// TIA Portal V19 export
FUNCTION "AutoAndResetTank" : Void   // FC56, STL
TITLE = Reset UHT
{ S7_Optimized_Access := 'TRUE' }
AUTHOR : OPA_8160
NAME : RESET
VERSION : 0.2
// ****** REVISION HISTORY :
// 
// VERSION DATE       BY  DESCRIPTION
// --------------------------------------------------------------------------
// 00.00               ORIGINAL FUNCTION BLOCK
// 
// 00.01 10/12 1997   OPA
//       FOLLOWING INSTRUCTIONS HAVE BEEN ADDED IN NETWORK 6
//       R     "S.T.01.REQUEST LYE"   "M242.0"     // STOP REQUESTING DETERGENT
//       R     "S.T.01.REQUEST ACID"  "M242.1"     // STOP REQUESTING DETERGENT
//       WITHOUT THESE TWO INSTRUCTIONS, DETERGENT PUMPS (LYE/ACID) COULD
//       CONTINUE DOSING AFTER STOP. 
// 00.02 11/2 1998    OPA   "S0 STOP CIP TANK" ADDED FOR "TANK AUTO"
// stored: AutoNumber false
BEGIN

NETWORK
TITLE = SET AUTO FLAG TANK
      O     "S0 PRESTERILIZING";
      O     "S0 STOP PRESTE. TANK";
      O     "S0 PRODUCTION TANK";
      O     "S0 STOP PRODUCTION TANK";
      O     "S0 CIP TANK";
      O     "S0 STOP CIP TANK";
      O     "S0 TOTAL STOP TANK";
      O     "LEDAssignment".SPARE_BUTTON1;

      =     "TANK AUTO";
      A     "LEDAssignment".SPARE_BUTTON1;

      R     "LEDAssignment".SPARE_BUTTON1;
      AN    "TANK AUTO";
      =     "M_AHV_SHUT_DOWN";
      AN    "S0 CIP TANK";
      JC    M001;
      A     "LowCIPPressure";
      JC    M003;  //"DB SETPOINTS".PT0167SpCIP
      A     "AcidCipPressure";
      JC    M004;
      L     "Setpoints".PT0167SpCIP;  // "DB SETPOINTS".PT0167SpCIPLow
      T     "STP_PT0167/IP0149_50".PT0167SpSTP;
      JU    M001;
M003: L     "Setpoints".PT0167SpCIPLow;
      T     "STP_PT0167/IP0149_50".PT0167SpSTP;
      JU    M001;
M004: L     "Setpoints".PT0167AcidPressure;
      T     "STP_PT0167/IP0149_50".PT0167SpSTP;

NETWORK
TITLE = FORCE VALVES TO AUTO
// THIS FORCE FUNCTION SETS ALL OUTPUTS IN AUTO MODE. I.E. VALVES, MOTORS, PUMPS 
// ETC.
M001: A     "TANK AUTO";
      FP    "ForceValves";
      JNB   M002;
      CALL  "Output Force to auto";
M002: NOP   0;

NETWORK
TITLE = RESET MANUAL MODE ON REGULATORS
// MAKE SURE THAT ALL RESET FROM AUTO, MANUAL, CASCADE OR FIXED MODE WHEN THE 
// PLANT 
// ENTER AUTO MODE
      AN    "TANK AUTO";
      FP    "UnforceValves";
      R     "AutoTT0172/IP0157";
      R     "ManTT0172/IP0157";
      R     "AutoPT0167/IP0149";
      R     "ManPT0167/IP0149";

NETWORK
TITLE = SET DUMMY RESET TANK
// THE FOLLOWING NETWORKS WILL RESET THE UHT-PLANT IF THE "UHT AUTO" FLAG 
// DISAPPEARS!
// I.E. PREPARE TOTAL STOP
      A     "TANK AUTO";
      S     "DUMMY RESET TANK";
      BEC;
      AN    "DUMMY RESET TANK";
      BEC;
      R     "DUMMY RESET TANK";

NETWORK
TITLE = RESET MAIN FLAGS FOR ALL DIFFERENT TANK-PROGRAM STEPS
      SET;
      R     "S0 STOP PRESTE. TANK";
      R     "S0 PRESTERILIZING";
      R     "S0 PRODUCTION TANK";
      R     "S0 STOP PRODUCTION TANK";
      R     "S0 TOTAL STOP TANK";
      R     "S0 CIP TANK";
      R     "S16 CIP TANK";

NETWORK
TITLE = RESET LED'S ON OPERATORPANEL
      R     "TANK STERILE";
      R     "TANK INITIALIZED";
      R     "LEDAssignment".K1_FLASH;  //"FLASH_K1_SPARE"
      R     "LEDAssignment".K1_LIGHT;  //"LIGHT_K1_SPARE"
      R     "LEDAssignment".K2_FLASH;  //"FLASH_K2_SPARE"
      R     "LEDAssignment".K2_LIGHT;  //"LIGHT_K2_SPARE"
      R     "LEDAssignment".K3_FLASH;  //"FLASH_K3_PRESTE."
      R     "LEDAssignment".K3_LIGHT;  //"LIGHT_K3_PRESTE."
      R     "LEDAssignment".K4_FLASH;  //"FLASH_K4_CIP_LYE"
      R     "LEDAssignment".K4_LIGHT;  //"LIGHT_K4_CIP_LYE"
      R     "LEDAssignment".K5_FLASH;  //"FLASH_K5_CIP_LYE_ACID"
      R     "LEDAssignment".K5_LIGHT;  //"LIGHT_K5_CIP_LYE_ACID"
      R     "LEDAssignment".K6_FLASH;  //"FLASH_K6_DRAIN_TANK"
      R     "LEDAssignment".K6_LIGHT;  //"LIGHT_K6_DRAIN_TANK"
      R     "LEDAssignment".K7_FLASH;  //"FLASH_K7_STOP"
      R     "LEDAssignment".K7_LIGHT;  //"LIGHT_K7_STOP"
//      R     M     57.6
//      R     M     57.7
      L     2#0000_0000_0000_0000;
//      T     MW    48                    // F-PUSHBUTTONS
//      T     MW    50                    // LED'S F-KEYS ON OPERATORPANEL
//      T     MW    52                    // LED'S F-KEYS ON OPERATORPANEL
//      T     MW    54                    // K-PUSHBUTTONS
      T     "Tag_88";  // TIMER UPDATE
      T     "Tag_89";  // AGITATOR, HELP FLAGS
      T     "Tag_90";  // DUMMIES
      R     "S.T.01.REQUEST LYE";  // STOP REQUESTING DETERGENT
      R     "S.T.01.REQUEST ACID";  // STOP REQUESTING DETERGENT

NETWORK
TITLE = RESET FLAGS AND DATA BIT FOR OUTPUTS
// //      L     0
// //      T     MD   246
// //      T     MD   250
// //
//       CALL  "STD_RESET_DATA_BIT"
//        DATABLOCK    :="ItemCommand"
//        START_WORD   :=0
//        LAST_WORD    :=96
//        BITS_TO_RESET:=W#16#1000

NETWORK
TITLE = Reset timer
// MAKE SURE THE RIGHT MESSAGE WILL APPEAR ON THE FIXED SCREEN OFF THE 
// OPERATORPANEL WHEN THE PLANT IS SWITCHED OFF.
      SET;
      L     0;
      T     "mw212_DW";
      T     "OP25 TANK".TaMainUpdating;
      T     "OP25 TANK".TaStepUpdating;
      T     "OP25 TANK".TaTimerStep;
      T     "OP25 TANK".TaTimerActual;
//RESET ALL TIMERS. THIS IS TO AVOID REMAINING TIME COUNTING ON THE FIXED
//SCREEN IN CASE OF RESTART
      R     "T 14 STERILE TIME";
      R     "T 15 COOLING TIME";
      R     "T 16 BLOW OUT COND";
      R     "T 17 BLOW OUT STOP";
      R     "T 18 DELAY 01.12";
      R     "T 27 WATER 1";
      R     "T 28 DOSING LYE";
      R     "T 29 LYE CIRCULATION";
      R     "T 30 WATER 2";
      R     "T 31 DOSING ACID";
      R     "T 32 ACID CIRCULATION";
      R     "T 33 WATER 3";
      R     "T 34 BLOW OUT CIP";
      R     "T 35 DELAY PT 01.67";
      R     "T 36 DELAY TT 01.76";
      R     "T 37 DELAY TT 01.78";
      R     "T 39 RUN 01.30";
      R     "T 44 FILLING DRAIN";
END_FUNCTION
